TYPE ST_EL7201 :
STRUCT
    sTerminalName : STRING(80) := 'EL7201-9014 | 1-Channel Servomotor';

    stTerminalInfo : ST_Terminal_Info;
	
	
	
END_STRUCT
END_TYPE

(* stored: Version 1.1.0.1, ProductVersion 3.1.4026.18
   DUT ST_EL7201: Id {33ba0efc-9fd3-4429-89c9-68e70c85eb6a} *)
